// TIA Portal V17 export
// export: Created 2024-09-27T18:48:48.3491252Z, ExportSetting WithDefaults, DisplayName Totally Integrated Automation Portal, DisplayVersion V17, DisplayName TIA Portal Openness, DisplayVersion V17, DisplayName TIA Portal Version Control Interface, DisplayVersion V17, DisplayName STEP 7 Professional, DisplayVersion V17, DisplayName STEP 7 Safety, DisplayVersion V17, DisplayName WinCC Professional, DisplayVersion V17
DATA_BLOCK "MC_MoveJog_DB_1"   // DB16
// stored: AutoNumber true, DBAccessibleFromOPCUA true, InstanceOfName MC_MoveJog, OfSystemLibElement MC_MoveJog, OfSystemLibVersion 8.0
"MC_MoveJog"
   // VAR_INPUT
   //    Axis : TO_SpeedAxis;
   //    JogForward : Bool;
   //    JogBackward : Bool;
   //    Velocity : Real;
   //    PositionControlled : Bool;
   // END_VAR
   // VAR_OUTPUT
   //    InVelocity : Bool;
   //    Busy : Bool;
   //    CommandAborted : Bool;
   //    Error : Bool;
   //    ErrorID : Word;
   //    ErrorInfo : Word;
   // END_VAR
   // VAR
   //    FB_ID : DInt;
   // END_VAR
BEGIN
END_DATA_BLOCK
